{attribute 'linkalways'} 
{attribute 'no_explicit_call' := 'This FB is a CLASS and must be accessed using methods or properties'}
{attribute 'enable_dynamic_creation'}
FUNCTION_BLOCK Node_F_VN_KeyPointsAndDescriptorsKAZEExp EXTENDS VisionNode
VAR
    ipSrcImage : _ITcVnImage;
    ipKeyPoints : _ITcVnContainer;
    ipDescriptors : _ITcVnImage;
    ipMask : _ITcVnImage;
    stParams : _TcVnParamsKAZE;
    hrPrev : _HRESULT(S_OK);
	hresult : _HRESULT(S_OK);
END_VAR

METHOD PUBLIC  Clone : I_Node
VAR
	pNode : POINTER TO Node_F_VN_KeyPointsAndDescriptorsKAZEExp;
END_VAR
pNode := __NEW(Node_F_VN_KeyPointsAndDescriptorsKAZEExp);
Clone := pNode^;
END_METHOD

METHOD FB_init : BOOL
VAR_INPUT
	bInitRetains : BOOL; // if TRUE, the retain variables are initialized (warm start / cold start)
	bInCopyCode : BOOL;  // if TRUE, the instance afterwards gets moved into the copy code (online change)
END_VAR
AddInput('ipSrcImage', ipSrcImage);
AddInput('ipMask', ipMask);
AddInput('stParams', stParams);
AddInput('hrPrev', hrPrev);
AddOutput('ipKeyPoints', ipKeyPoints);
AddOutput('ipDescriptors', ipDescriptors);
AddOutput('hresult',hresult);
END_METHOD

METHOD PROTECTED OnExecute
hresult.Value := F_VN_KeyPointsAndDescriptorsKAZEExp(
	ipSrcImage := ipSrcImage.Value,
    ipKeyPoints := ipKeyPoints.Value,
    ipDescriptors := ipDescriptors.Value,
    ipMask := ipMask.Value,
    stParams := stParams.Value,
	hrPrev:= hrPrev.Value);
END_METHOD

METHOD PUBLIC PreExecutionCheck
VAR_INPUT
	Check : I_PreExecutionChecks;
END_VAR
Check.IsTrue(ipSrcImage.IsValid, 'ipSrcImage must contain an image');
Check.IsTrue(ipSrcImage.HasChannelCount(1), 'ipSrcImage must have 1 channel');
END_METHOD

END_FUNCTION_BLOCK

(* stored: Version 1.1.0.1, ProductVersion 3.1.4024.15
   POU Node_F_VN_KeyPointsAndDescriptorsKAZEExp: Id {22a0ffb6-13f4-0dcb-0685-d934bb96aee2}, SpecialFunc None
   Folder Constructor: Id {2090cf7e-13a0-0fa2-00f1-99afd6697ed1}
   Method Clone: Id {0f6129ac-cf88-0c9f-258b-63e04b8180a8}
   Method FB_init: Id {4b2175d8-b1f5-0b93-2fef-f7beddcb9dc7}
   Method OnExecute: Id {3c758cf5-d083-0410-154e-fb092c4136c5}
   Method PreExecutionCheck: Id {29bbdbe8-dcf0-0fe5-1d18-60fcdd40e94c} *)
